FUNCTION_BLOCK TTestEventHandler_UsesEventArgs IMPLEMENTS ITestEventHandler_UsesEventArgs
VAR
    _EventWasRaised : BOOL;
    Arg1 : UDINT;
    Arg2 : LREAL;
    Arg3 : STRING;
    Arg4 : T_MAxString;
    Arg5 : BOOL;
END_VAR

PROPERTY EventWasRaised : BOOL
GET
EventWasRaised := _EventWasRaised;
END_GET
END_PROPERTY

METHOD OnThisEvent
VAR_INPUT
    EventArgs : IStreamReader;
END_VAR
Arg1 := EventArgs.Read_UDINT();
Arg2 := EventArgs.Read_LREAL();
Arg3 := EventArgs.Read_String();
Arg4 := EventArgs.Read_STRING();
Arg5 := EventArgs.Read_BOOL();

_EventWasRaised := TRUE;
END_METHOD

END_FUNCTION_BLOCK

(* stored: Version 1.1.0.1, ProductVersion 3.1.4024.4
   POU TTestEventHandler_UsesEventArgs: Id {68a56228-f403-4fd1-b44e-660934df017d}, SpecialFunc None
   Property EventWasRaised: Id {61cb43d3-da0e-43c2-9c68-d0552570ec9b}
   Get Get: Id {9d6b8bdb-5d44-441a-8270-cd1801f2ebc1}
   Method OnThisEvent: Id {ec32bc6f-ebed-4901-a0ea-d9a86aacf099} *)
